PROGRAM P_feedback_calculation
VAR
END_VAR

(*
 *************************************************************************************************************
 * \file  P_feedback_calc
 * \author Quique
 * \version 1.0.0
 * \date Creation: 16/07/2021
 * \brief Selects P used in feedback 
 *************************************************************************************************************
 \defgroup P_CONTROL - FEEDBACK_CALC
 
 \brief 	This algorithm is used to determine which is the phase with the less power consumption and then
 			this obtained value is used as the feedback of P loop. The goal is that this value
			is updated continuously to guarantee that there is null P injection to grid during stationary
			regime. 
		
 \details 	This algorithm is based on a first order approach assuming that line power equals the summatory 
			of 3 single - phase powers. Thus and since it is mandatory to not inject P to grid, the algorithm
			checks which is the phase with the less consumption value, multiplies it by three 

*)

//Determination of P_measured_min
Min_P_calculation();

//  Ploop in closed loop
IF NOT GVL_P_CONTROL.P_loop_type THEN
	GVL_P_CONTROL.P_feedback:= GVL_POWERMETER.P_min;
ELSE
// Ploop in open loop	
	GVL_P_CONTROL.P_feedback:= GVL_POWERMETER.P_pu;
END_IF

END_PROGRAM

(* stored: Version 1.1.0.1, ProductVersion 3.1.4024.11
   POU P_feedback_calculation: Id {b7ec539d-9ec1-4c87-b13f-1b2639dff2a3}, SpecialFunc None *)
